// TIA Portal V20 export
// export: Created 2025-12-01T14:56:09.353886Z, ExportSetting None, DisplayName Totally Integrated Automation Portal, DisplayVersion V20 Update 3, DisplayName TIA Portal Openness, DisplayVersion V20 Update 3, DisplayName TIA Portal Version Control Interface, DisplayVersion V20 Update 3, DisplayName STEP 7 Professional, DisplayVersion V20 Update 3, DisplayName STEP 7 Safety, DisplayVersion V20 Update 2, DisplayName WinCC Basic/Comfort/Advanced, DisplayVersion V20 Update 3, DisplayName WinCC Professional, DisplayVersion V20 Update 3, DisplayName WinCC Unified, DisplayVersion V20 Update 3
TYPE "UDT_DatosGalibo"
   STRUCT
      Codigo : Struct
         Galibo : Word;
         HuecoTaco : Word;
         GaliboExtra : Word;
      END_STRUCT;
      GaliboAltura : USInt;   // Galibo --> Altura
      GaliboAnchura : USInt;   // Galibo --> Anchura
      GaliboProfundidad : USInt;   // Galibo --> Profuncidad
      GaliboTaco : USInt;   // Galibo --> Taco
      GaliboHueco : USInt;   // Galibo --> Hueco
      GaliboHuecoRemontado : USInt;   // Galibo --> Hueco Remontada
      GaliboColor : USInt;   // Galibo --> Color
      GaliboPatin : USInt;   // Galibo --> Patin
      GaliboTipoCarga : USInt;   // Galibo --> Tipo de Carga (Euro,Caja...)
      GaliboRemontada : USInt;   // Galibo --> Carga remontada
      GaliboVacia : USInt;   // Galibo --> Carga Vacia
      CotaAltura : UInt;   // Cota de Altura de la UT
      CotaAnchura : UInt;   // Cota de Anchura de la UT
      CotaProfundidad : UInt;   // Cota de Profundidad de la UT
      Peso : UDInt;   // Peso de la UT
      EtiquetaRouter : UDInt;
   END_STRUCT;
END_TYPE
